// TIA Portal V19 export
TYPE "LEXCHANGETRAY_typeXXXIoSignalContronNodeMonitoring"
// stored: Access Published
   STRUCT
      simulated : Bool;
      u1CellsSignal1 : Bool;
      u1CellsSignal2 : Bool;
      u1CellsSignal3 : Bool;
      u1CellsSignal4 : Bool;
      u2CellsSignal1 : Bool;
      u2CellsSignal2 : Bool;
      u2CellsSignal3 : Bool;
      u2CellsSignal4 : Bool;
      ngStrapSignal : Bool;
      ngSafeDoorSignal : Bool;
      ngMateriaFullSignal : Bool;
      beltForwardButton : Bool;
      beltBackForwardButton : Bool;
   END_STRUCT;
END_TYPE
